Fanuc KAREL source: kt00519.KL

-- PROVISIONAL review KL for V1013-1; original PC SHA256 774117148ae956f29f75a788a26f9940dd037849fbaab3a3a4b874ae72904fe0
-- Incomplete behavior may be omitted. Consult companion uncertainty JSON. Do not deploy.
PROGRAM KT00519
%NOLOCKGROUP
-- UNRESOLVED_DECL P1 type=000106
-- UNRESOLVED_DECL P2 type=000102
-- UNRESOLVED_DECL OUT type=000101
BEGIN
  -- UNRESOLVED_PC offsets 5-20; opcodes 2E,22,32,35
  -- UNRESOLVED_PC offsets 25-40; opcodes 2E,22,32,35
  -- UNRESOLVED_PC offsets 45-79; opcodes 49,7E,49,7E,60,4A
  -- UNRESOLVED_PC offsets 84-88; opcodes 7F
END KT00519
